FUNCTION_BLOCK OR_10 (* FB to calculate bitwise boolean OR (generic FB) *)
  (* Standard: 61131-3; Classification: standard bitwise boolean function; Description: Copyright (c) 2014 Profactor GmbH This program and the accompanying materials are made available under the terms of the Eclipse Public License 2.0 which is available at https://www.eclipse.org/legal/epl-2.0/ SPDX-License-Identifier: EPL-2.0 *)
  (* Version 3.0, 2025-04-14, Patrick Aigner, changed package *)
  (* Version 1.0, 2014-10-11, Matthias Plasch, Profactor GmbH *)
  PACKAGE iec61131::bitwiseOperators;
  {SET_ATTRIBUTE(eclipse4diac::core::GenericClassName, 'GEN_OR')}
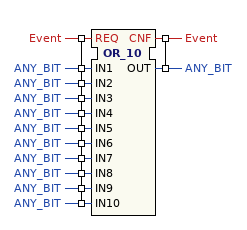
  EVENT_INPUT
    REQ WITH IN1, IN2, IN3, IN4, IN5, IN6, IN7, IN8, IN9, IN10; (* Normal Execution Request *)
  END_EVENT
  EVENT_OUTPUT
    CNF WITH OUT; (* Execution Confirmation *)
  END_EVENT
  VAR_INPUT
    IN1 : ANY_BIT; (* OR input 1 *)
    IN2 : ANY_BIT; (* OR input 2 *)
    IN3 : ANY_BIT; (* OR input 3 *)
    IN4 : ANY_BIT; (* OR input 4 *)
    IN5 : ANY_BIT; (* OR input 5 *)
    IN6 : ANY_BIT; (* OR input 6 *)
    IN7 : ANY_BIT; (* OR input 7 *)
    IN8 : ANY_BIT; (* OR input 8 *)
    IN9 : ANY_BIT; (* OR input 9 *)
    IN10 : ANY_BIT; (* OR input 10 *)
  END_VAR
  VAR_OUTPUT
    OUT : ANY_BIT; (* OR result *)
  END_VAR
END_FUNCTION_BLOCK
